PROGRAM historical
VAR
	
	state: INT;
END_VAR




CASE state OF

0:	
IF gvl.bHistory THEN
	CASE gvl.radioEstufa OF
0:
	IF gvl.radioFiltro = 0 THEN
		state:=10;
	gvl.sCmdSelect19:= 'SELECT [data],[hora],[auto],[pos],[OF],[lote],[class],[pot],[isola],[fPot],[reator],[time],[temp] FROM [dbo].[ProcessTable19] 
	WHERE data=$'';
	gvl.sCmdSelect19:= concat(gvl.sCmdSelect19,gvl.arrCVSfilter[0].ano);
	gvl.sCmdSelect19:= concat(gvl.sCmdSelect19,'-');
	gvl.sCmdSelect19:= concat(gvl.sCmdSelect19,gvl.arrCVSfilter[0].mes);
	gvl.sCmdSelect19:= concat(gvl.sCmdSelect19,'-');
	gvl.sCmdSelect19:= concat(gvl.sCmdSelect19,gvl.arrCVSfilter[0].dia);
	gvl.sCmdSelect19:= concat(gvl.sCmdSelect19,'$';');
	ELSIF gvl.radioFiltro = 1 THEN
		state:=10;
	gvl.sCmdSelect19:= 'SELECT [data],[hora],[auto],[pos],[OF],[lote],[class],[pot],[isola],[fPot],[reator],[time],[temp] FROM [dbo].[ProcessTable19] 
	WHERE OF=$'';
	gvl.sCmdSelect19:= concat(gvl.sCmdSelect19,gvl.arrCVSfilter[0].ordem);
	gvl.sCmdSelect19:= concat(gvl.sCmdSelect19,'$';');
	ELSIF gvl.radioFiltro = 2 THEN
		state:=10;
	gvl.sCmdSelect19:= 'SELECT [data],[hora],[auto],[pos],[OF],[lote],[class],[pot],[isola],[fPot],[reator],[time],[temp] FROM [dbo].[ProcessTable19] 
	WHERE lote=$'';
	gvl.sCmdSelect19:= concat(gvl.sCmdSelect19,gvl.arrCVSfilter[0].lote);
	gvl.sCmdSelect19:= concat(gvl.sCmdSelect19,'$';');
	END_IF
	
1:
	IF gvl.radioFiltro = 0 THEN
		state:=10;
	gvl.sCmdSelect19:= 'SELECT [data],[hora],[auto],[pos],[OF],[lote],[class],[pot],[isola],[fPot],[reator],[time],[temp] FROM [dbo].[ProcessTable20] 
	WHERE data=$'';
	gvl.sCmdSelect19:= concat(gvl.sCmdSelect19,gvl.arrCVSfilter[0].ano);
	gvl.sCmdSelect19:= concat(gvl.sCmdSelect19,'-');
	gvl.sCmdSelect19:= concat(gvl.sCmdSelect19,gvl.arrCVSfilter[0].mes);
	gvl.sCmdSelect19:= concat(gvl.sCmdSelect19,'-');
	gvl.sCmdSelect19:= concat(gvl.sCmdSelect19,gvl.arrCVSfilter[0].dia);
	gvl.sCmdSelect19:= concat(gvl.sCmdSelect19,'$';');
	ELSIF gvl.radioFiltro = 1 THEN
		state:=10;
	gvl.sCmdSelect19:= 'SELECT [data],[hora],[auto],[pos],[OF],[lote],[class],[pot],[isola],[fPot],[reator],[time],[temp] FROM [dbo].[ProcessTable20] 
	WHERE OF=$'';
	gvl.sCmdSelect19:= concat(gvl.sCmdSelect19,gvl.arrCVSfilter[0].ordem);
	gvl.sCmdSelect19:= concat(gvl.sCmdSelect19,'$';');
	ELSIF gvl.radioFiltro = 2 THEN
		state:=10;
	gvl.sCmdSelect19:= 'SELECT [data],[hora],[auto],[pos],[OF],[lote],[class],[pot],[isola],[fPot],[reator],[time],[temp] FROM [dbo].[ProcessTable20] 
	WHERE lote=$'';
	gvl.sCmdSelect19:= concat(gvl.sCmdSelect19,gvl.arrCVSfilter[0].lote);
	gvl.sCmdSelect19:= concat(gvl.sCmdSelect19,'$';');
	END_IF
	
2:
	IF gvl.radioFiltro = 0 THEN
		state:=10;
	gvl.sCmdSelect19:= 'SELECT [data],[hora],[auto],[pos],[OF],[lote],[class],[pot],[isola],[fPot],[reator],[time],[temp] FROM [dbo].[ProcessTable21] 
	WHERE data=$'';
	gvl.sCmdSelect19:= concat(gvl.sCmdSelect19,gvl.arrCVSfilter[0].ano);
	gvl.sCmdSelect19:= concat(gvl.sCmdSelect19,'-');
	gvl.sCmdSelect19:= concat(gvl.sCmdSelect19,gvl.arrCVSfilter[0].mes);
	gvl.sCmdSelect19:= concat(gvl.sCmdSelect19,'-');
	gvl.sCmdSelect19:= concat(gvl.sCmdSelect19,gvl.arrCVSfilter[0].dia);
	gvl.sCmdSelect19:= concat(gvl.sCmdSelect19,'$';');
	ELSIF gvl.radioFiltro = 1 THEN
		state:=10;
	gvl.sCmdSelect19:= 'SELECT [data],[hora],[auto],[pos],[OF],[lote],[class],[pot],[isola],[fPot],[reator],[time],[temp] FROM [dbo].[ProcessTable21] 
	WHERE OF=$'';
	gvl.sCmdSelect19:= concat(gvl.sCmdSelect19,gvl.arrCVSfilter[0].ordem);
	gvl.sCmdSelect19:= concat(gvl.sCmdSelect19,'$';');
	ELSIF gvl.radioFiltro = 2 THEN
		state:=10;
	gvl.sCmdSelect19:= 'SELECT [data],[hora],[auto],[pos],[OF],[lote],[class],[pot],[isola],[fPot],[reator],[time],[temp] FROM [dbo].[ProcessTable21] 
	WHERE lote=$'';
	gvl.sCmdSelect19:= concat(gvl.sCmdSelect19,gvl.arrCVSfilter[0].lote);
	gvl.sCmdSelect19:= concat(gvl.sCmdSelect19,'$';');
	END_IF
	END_CASE
ELSE
	state:=0;	
END_IF

10:
IF NOT main.bBusySelect19 THEN
	state:=20;
	gvl.bSelect19:= TRUE;
ELSE
	state:=10;
END_IF

20:
IF NOT main.bBusySelect19 THEN
	state:=30;
	gvl.bSelect19:= FALSE;
	P_TextModeWrite.bWrite:= TRUE;
ELSE
	state:=20;
END_IF

30:
IF NOT P_TextModeWrite.bBusy AND not P_TextModeWrite.bWrite THEN
	state:=0;
	gvl.bHistory:=FALSE;
ELSE
	state:=30;
END_IF

END_CASE

END_PROGRAM

(* stored: Version 1.1.0.1, ProductVersion 3.1.4024.12
   POU historical: Id {81f57b33-e15a-4aed-8714-0c721fd5b1e9}, SpecialFunc None *)
